// TIA Portal V18 export
FUNCTION_BLOCK "System_Enable"   // FB15, LAD
{ S7_Optimized_Access := 'TRUE' }
// Written BY Kristopher Gimenez January 26,2023
// This block is used to control enable the Pump and Fail safe valves based on HPU Startup.
// stored: AutoNumber false, MemoryReserve 100, SetENOAutomatically false
BEGIN

REGION Network 1: Enable System
   // Turn On Pump Enable and Fail save if Pumps have started or tried and are off ,with an elec HPU. 
   // Turn On Pump Enable and Fail Save if StartCAt
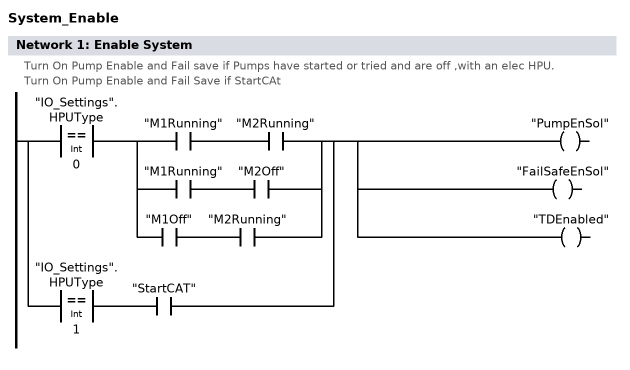
   RUNG wire#powerrail
      { S7_Templates := "SrcType := Int" } EQ_Contact(in1 := "IO_Settings".HPUType, in2 := 0)
      wire#w1
      Contact( "M1Running" )
      Contact( "M2Running" )
      wire#w2
      Coil( "PumpEnSol" )
   END_RUNG
   RUNG wire#w1
      Contact( "M1Running" )
      Contact( "M2Off" )
   END_RUNG wire#w2
   RUNG wire#w1
      Contact( "M1Off" )
      Contact( "M2Running" )
   END_RUNG wire#w2
   RUNG wire#powerrail
      { S7_Templates := "SrcType := Int" } EQ_Contact(in1 := "IO_Settings".HPUType, in2 := 1)
      Contact( "StartCAT" )
   END_RUNG wire#w2
   RUNG wire#w2
      Coil( "FailSafeEnSol" )
   END_RUNG
   RUNG wire#w2
      Coil( "TDEnabled" )
   END_RUNG
   // the same network as SCL:
   "PumpEnSol" := (("IO_Settings".HPUType = 0) AND (("M1Running" AND "M2Running") OR ("M1Running" AND "M2Off") OR ("M1Off" AND "M2Running"))) OR (("IO_Settings".HPUType = 1) AND "StartCAT");
   "FailSafeEnSol" := "PumpEnSol";
   "TDEnabled" := "PumpEnSol";
END_REGION
END_FUNCTION_BLOCK
